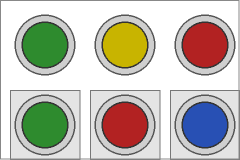
VISUALIZATION VIS_Main  // 240x160
    Lamp1 (10,10 70x70), variable: gHMI.Run, style: Lamp-Lamp1-Green
    Lamp1 (90,10 70x70), variable: gHMI.Alarm, style: Lamp-Lamp1-Yellow
    PushSwitch (10,90 70x70), variable: gHMI.Start, behaviour: TAP, style: Switch-PushSwitch-Green
    PushSwitch (90,90 70x70), variable: gHMI.Stop, behaviour: TAP, style: Switch-PushSwitch-Red
    PushSwitch (170,90 70x70), variable: gHMI.Reset, behaviour: TAP, style: Switch-PushSwitch-Blue
    Lamp1 (170,10 70x70), variable: gHMI.Error, style: Lamp-Lamp1-Red
END_VISUALIZATION

(* stored: Version 1.1.0.1, ProductVersion 3.1.4024.12
   Visu VIS_Main: Id {423f1b75-2deb-4e31-b614-a24bd0155a9f} *)
